(* CODESYS project CodeSys_Demo1

Project tree, tasks and I/O mapping:
  Device : CODESYS Control Win V3 x64, CODESYS, version 3.5.20.20
    application Application
      libraries: Standard, 3.5.18.0 (System)
      task MainTask (cyclic, interval t#20ms, priority 1) calls PLC_PRG
      global variables OPCUA_DB1
      program PLC_PRG [ST]
      Symbols
*)

// Device/Application/OPCUA_DB1
{attribute 'qualified_only'}
VAR_GLOBAL
	iStart: BOOL;
	iStop: BOOL;
	oRun: BOOL;
END_VAR

// Device/Application/PLC_PRG
PROGRAM PLC_PRG
VAR
END_VAR

END_PROGRAM
